// TIA Portal V18 export
DATA_BLOCK "FB1-MR_Flowrate Control_DB"   // DB39
VERSION : 0.1
// stored: AutoNumber true, DBAccessibleFromOPCUA true, InstanceOfName FB1-MR_Flowrate Control, InstanceOfType FB
"FB1-MR_Flowrate Control"
   // VAR_INPUT
   //    "Pump size A" : Real;
   //    "pump size B" : Real;
   //    "Pump speed A" : Real;
   //    "pump Speed B" : Real;
   //    "Mixing Ratio 100:B" : Real;
   //    "Metering Qty" : Real;
   //    "Metering Flowrate" : Real;
   //    "Flowrate Adjustemnt A %" : Real;
   //    "Flowrate Adjustment B %" : Real;
   //    "Pump A max Hz" : Real;
   //    "pump B max Hz" : Real;
   // END_VAR
   // VAR_OUTPUT
   //    "Flowrate pump A without adjustment" : Real;
   //    "Flowrate pump B without adjustment" : Real;
   //    "Flowrate pump A with adjustment" : Real;
   //    "Flowrate pump B with adjustment" : Real;
   //    "Mixed Flowrate" : Real;
   //    "Pump Capacity A cc/min" : Real;
   //    "Pump capacity B cc/min" : Real;
   //    "Pump A frequency" : Real;
   //    "Pump B frequency" : Real;
   //    "Metering time" : DInt;
   //    "Meteringtime in sec" : Int;
   // END_VAR
   // VAR
   //    "Maximum Flowrate Pump A" : Real;
   //    "Maximum Flowrate Pump B" : Real;
   //    "Pump compensation" : Real;
   //    "Individual flowrate A MR" : Real;
   //    "Individual flowrate B1 MR" : Real;
   //    "Individual flowrate B MR" : Real;
   //    "Flowrate Ratio difference A" : Real;
   //    "Flowrate Ratio difference B" : Real;
   //    "Flowrate Pump A" : Real;
   //    "Flowrate Pump B" : Real;
   //    "Flowrate B After Compensation" : Real;
   //    "Mixed flowrate A+B" : Real;
   //    "Flowrate to adjust A" : Real;
   //    "Flowrate to adjust B" : Real;
   //    "metering time in minutes" : Real;
   //    "metering time in Sec" : Real;
   //    "Metering time in msec" : LReal;
   //    "flowrate to adjust A_1" : Real;
   //    "flowrate to adjust B_1" : Real;
   //    "Ratio>100" : Real;
   //    "amount to reduce in A" : Real;
   //    "Flowrate difference" : Real;
   //    "Ratio margin" : Real;
   //    "Ratio/100" : Real;
   //    "Flowrate A Per ratio" : Real;
   //    "A Flowrate Compensated" : Real;
   // END_VAR
BEGIN
END_DATA_BLOCK
